Staubli VAL3: setupRosMsgs.pgx

public program setupRosMsgs()
begin
  // Robot status message
  //rosMsgStatus.header.nMsgType=13
  //rosMsgStatus.header.nCommType=1
  //rosMsgStatus.header.nReplyCode=0

  // Joint trajectory point message
  //rosMsgJointTraj.header.nMsgType=14
  //rosMsgJointTraj.header.nCommType=1
  //rosMsgJointTraj.header.nReplyCode=0

  // Feedback of joint position/velocity/acceleration
  // prefix length = 12 + 132 = 144
  //rosMsgJointFbk.prefix.nLength=144
  //rosMsgJointFbk.header.nMsgType=15
  //rosMsgJointFbk.header.nCommType=1
  //rosMsgJointFbk.header.nReplyCode=0

  // robot_id
  //rosMsgJointFbk.body.nData[0] = 0
  // valid_fields
  //rosMsgJointFbk.body.nData[1] = 2
  // time
  //rosMsgJointFbk.body.nData[2] = 3.2


  // Feedback of joint position
  // prefix length = 12 + 44
  rosMsgJointFbk.prefix.nLength=56
  rosMsgJointFbk.header.nMsgType=10
  rosMsgJointFbk.header.nCommType=1
  rosMsgJointFbk.header.nReplyCode=0
  // sequence
  rosMsgJointFbk.body.nData[0] = 0
end
